FUNCTION_BLOCK FB_TransportLogik
VAR_INPUT
	bEnable : BOOL;
	bExecute : BOOL;
	eStateE : eBetriebszustand;
	nStation : INT;
	// Logik -> Hardware Signal
	bStation1 : BOOL;
	bStation2 : BOOL;
	bStation3 : BOOL;
	bStation4 : BOOL; 
END_VAR
VAR_OUTPUT
	bEnableA : BOOL;
	bExecuteA : BOOL;
	bStopA : BOOL;
	eStateA : eBetriebszustand;
	// Hardware Signale -> Logik
	bStop1 : BOOL;
	bStop2 : BOOL;
	bStop3 : BOOL;
	
 
END_VAR
VAR
	nState : INT;
END_VAR

CASE nState OF
	0: // OFF
	bEnableA := FALSE;
	bExecuteA := FALSE;
	bStopA := FALSE;
	eStateA := eBetriebszustand.Off;
	
	IF bEnable THEN
		nState := 1;
	END_IF
	
	1: //INIT
	bEnableA := TRUE;
	bExecuteA := FALSE;
	bStopA := FALSE;
	
	IF eStateE = eBetriebszustand.Ready THEN
		nState := 2; // Ready
	END_IF
	
	2: // READY
	bEnableA := TRUE;
	bExecuteA := FALSE;
	bStopA := FALSE;
	
	IF bExecute THEN
		nState := 3;
	END_IF
	
	3: // FB TransportBand start
	bExecuteA := TRUE;
	
	IF (nStation - 1) = 1 THEN
		bStop1 := FALSE;
	ELSIF (nStation - 1) = 2 THEN
		bStop2 :=FALSE;
	ELSIF (nStation - 1) = 3 THEN
		bStop3 := FALSE;
	END_IF
	
	IF bStation1 AND (nStation = 1) THEN
		nState := 4;
	ELSIF bStation2 AND (nStation = 2) THEN
		nState := 4;
	ELSIF bStation3 AND (nStation = 3) THEN
		nState := 4;
	ELSIF bStation4 AND (nStation = 4) THEN
		nState := 4;
	END_IF
	
	4: // TransportBand Stop
	
	bExecuteA := FALSE;
	bStopA := TRUE;
	
	IF (nStation - 1) = 1 THEN
		bStop1 := TRUE;
	ELSIF (nStation - 1) = 2 THEN
		bStop2 := TRUE;
	ELSIF (nStation - 1) = 3 THEN
		bStop3 := TRUE;
	END_IF
	
	IF eStateE = eBetriebszustand.Done THEN
		nState := 5;
	END_IF
	
	5: // DONE
	eStateA := eBetriebszustand.Done;
	
	IF NOT bExecute THEN
		nState := 2;
	END_IF
	
	
	
	
END_CASE

END_FUNCTION_BLOCK

(* stored: Version 1.1.0.1, ProductVersion 3.1.4024.15
   POU FB_TransportLogik: Id {d1820bad-b280-4a8e-a997-4a6fae8b8423}, SpecialFunc None *)
